FUNCTION_BLOCK INCHOICE (* Composite Function Block Type *)
  (* Standard: 61499-2 *)
  (* Version 0.0, 09/08/2022, Pranay Jhunjhunwala, Schneider Electric, template *)
  PACKAGE Main;
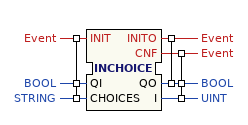
  EVENT_INPUT
    INIT WITH QI, CHOICES; (* Initialization Request *)
  END_EVENT
  EVENT_OUTPUT
    INITO WITH QO; (* Initialization Confirm *)
    CNF WITH QO, I; (* Execution Confirmation *)
  END_EVENT
  VAR_INPUT
    QI : BOOL; (* Input event qualifier *)
    CHOICES : STRING;
  END_VAR
  VAR_OUTPUT
    QO : BOOL; (* Output event qualifier *)
    I : UINT;
  END_VAR
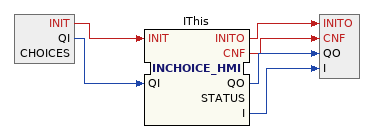
  FBS
    IThis : INCHOICE_HMI;
  END_FBS
  EVENT_CONNECTIONS
    INIT TO IThis.INIT;
    IThis.INITO TO INITO;
    IThis.CNF TO CNF;
  END_CONNECTIONS
  DATA_CONNECTIONS
    QI TO IThis.QI;
    IThis.I TO I;
    IThis.QO TO QO;
  END_CONNECTIONS
END_FUNCTION_BLOCK
